(* Schneider Machine Expert - Basic project Motor 3 fasa Delta Star, file version 1.7.0.0 *)
(* ProjectInformations: Name=New project *)

HARDWARE
  Cpu 0: TM221M16R/G
  EthernetConfiguration: NetworkName=M221, IpAllocationMode=FixedAddress, IpAddress=0.0.0.0, SubnetMask=0.0.0.0
  SerialLineConfiguration: Baud=Baud19200, Parity=ParityEven, DataBits=DataBits8, StopBits=StopBits1, PhysicalMedium=PhysicalMediumRs485, TransmissionMode=TransmissionModeModbusRtu, SlaveId=1, Addressing=SlaveAddressing
  MastTask: UsePeriodScanMode=false, PeriodScan=100
  FastTask: Period=255
  CpuBehavior: StartingMode=StartAsPreviousState, AutoSaveRamOnEeprom=true, WatchdogPeriod=250

SYMBOLS  (address, symbol, comment, settings)
  %TM0        [Preset=20, Base=OneHundredMilliSeconds]
  %TM1        [Preset=5, Base=OneSecond]

POU New POU
  (* SectionNumber=1 *)

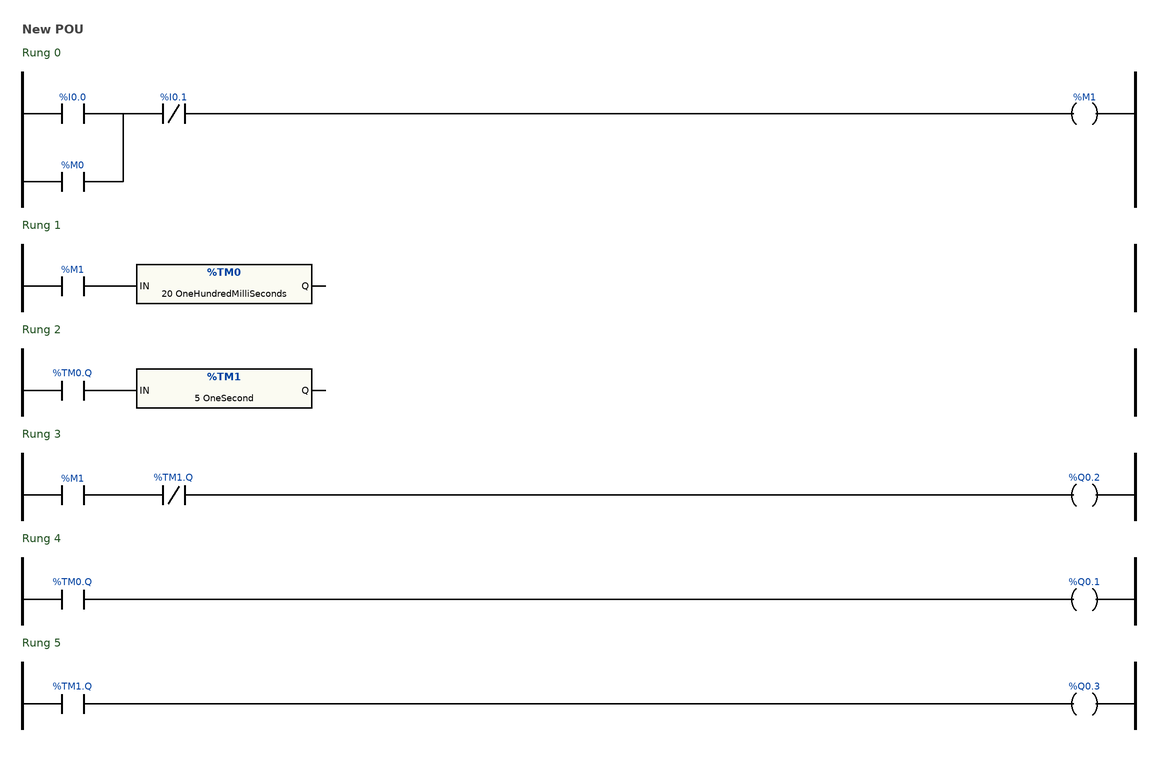

// Rung 0
  LD %I0.0
  OR %M0
  ANDN %I0.1
  ST %M1
  // as ST:
  //   %M1 := (%I0.0 OR %M0) AND NOT %I0.1;

// Rung 1
  BLK %TM0
  LD %M1
  IN
  END_BLK
  // as ST:
  //   %TM0(IN := %M1);

// Rung 2
  BLK %TM1
  LD %TM0.Q
  IN
  END_BLK
  // as ST:
  //   %TM1(IN := %TM0.Q);

// Rung 3
  LD %M1
  ANDN %TM1.Q
  ST %Q0.2
  // as ST:
  //   %Q0.2 := %M1 AND NOT %TM1.Q;

// Rung 4
  LD %TM0.Q
  ST %Q0.1
  // as ST:
  //   %Q0.1 := %TM0.Q;

// Rung 5
  LD %TM1.Q
  ST %Q0.3
  // as ST:
  //   %Q0.3 := %TM1.Q;
